{attribute 'linkalways'} 
{attribute 'no_explicit_call' := 'This FB is a CLASS and must be accessed using methods or properties'}
{attribute 'enable_dynamic_creation'}
FUNCTION_BLOCK Node_F_VN_ContourCircularity EXTENDS VisionNode
VAR
    ipContour : _ITcVnContainer;
    fCircularity : _LREAL(0.0);
    hrPrev : _HRESULT(S_OK);
	hresult : _HRESULT(S_OK);
END_VAR

METHOD PUBLIC  Clone : I_Node
VAR
	pNode : POINTER TO Node_F_VN_ContourCircularity;
END_VAR
pNode := __NEW(Node_F_VN_ContourCircularity);
Clone := pNode^;
END_METHOD

METHOD FB_init : BOOL
VAR_INPUT
	bInitRetains : BOOL; // if TRUE, the retain variables are initialized (warm start / cold start)
	bInCopyCode : BOOL;  // if TRUE, the instance afterwards gets moved into the copy code (online change)
END_VAR
AddInput('ipContour', ipContour);
AddInput('hrPrev', hrPrev);
AddOutput('fCircularity', fCircularity);
AddOutput('hresult',hresult);
END_METHOD

METHOD PROTECTED OnExecute
hresult.Value := F_VN_ContourCircularity(
	ipContour := ipContour.Value,
    fCircularity := fCircularity.Value,
	hrPrev:= hrPrev.Value);
END_METHOD

METHOD PUBLIC PreExecutionCheck
VAR_INPUT
	Check : I_PreExecutionChecks;
END_VAR
Check.IsTrue(ipContour.IsValid, 'ipContour must be a valid container');
Check.IsTrue((ipContour.IsType(TC_GLOBAL_CONST_LIST.ContainerType_Vector_TcVnPoint2_DINT) OR
              ipContour.IsType(TC_GLOBAL_CONST_LIST.ContainerType_Vector_TcVnPoint2_REAL)),
              'ipContour contains incorrect type');
END_METHOD

END_FUNCTION_BLOCK

(* stored: Version 1.1.0.1, ProductVersion 3.1.4026.13
   POU Node_F_VN_ContourCircularity: Id {4a72326e-5df5-0604-191b-1a52f989dfcc}, SpecialFunc None
   Folder Constructor: Id {10bddbc3-fc63-0c1e-2737-dee90bff2317}
   Method Clone: Id {198fb635-51f9-0012-2733-0276103cb807}
   Method FB_init: Id {eee07bb4-4547-0e1a-1653-45857b687610}
   Method OnExecute: Id {6344f807-590f-096f-0074-27268a060427}
   Method PreExecutionCheck: Id {23d0bd0c-3aff-0939-10c0-4e16adee5915} *)
